// TIA Portal project "SCL EJERCICIO 5" (V11)

(* hardware
DEVICE "S7300/ET200 station_1"  SIMATIC 300-Station
   slot 0: "Perfil soporte_0"  Rail  6ES7 390-1***0-0AA0
   slot 2: "PLC_1"  CPU 313C-2 DP  6ES7 313-6CF03-0AB0  V2.6
      slot 0: "Interfaz MPI_1"  MPI
      slot 1: "Interfaz DP_1"  DP
      slot 2: "DI16/DO16_1"  DI16/DO16
      slot 4: "Contaje_1"  Counter
*)

// ===== PLC "PLC_1"  CPU 313C-2 DP =====

VAR_GLOBAL   // PLC tag table "Tabla de variables estándar"
   "Tag_1" AT %E0.0 : Bool;
   "Tag_2" AT %E0.1 : Bool;
   "Tag_3" AT %E0.2 : Bool;
   "Tag_4" AT %E0.3 : Bool;
   "Tag_5" AT %E0.4 : Bool;
   "Tag_6" AT %E0.5 : Bool;
   "Tag_7" AT %E0.6 : Bool;
   "Tag_8" AT %E0.7 : Bool;
   "Tag_9" AT %E1.0 : Bool;
   "Tag_10" AT %E1.1 : Bool;
   "Tag_11" AT %A0.0 : Bool;
   "Tag_12" AT %A0.1 : Bool;
   "Tag_13" AT %A0.2 : Bool;
   "Tag_14" AT %A0.3 : Bool;
   "Tag_15" AT %A0.4 : Bool;
   "Tag_16" AT %A0.5 : Bool;
   "Tag_17" AT %A0.6 : Bool;
   "Tag_18" AT %A0.7 : Bool;
   "Tag_19" AT %A1.0 : Bool;
   "Tag_20" AT %A1.1 : Bool;
   "Tag_21" AT %M0.0 : Bool;
   "Tag_22" AT %MW10 : Int;
   "Tag_23" AT %A1.2 : Bool;
   "Tag_24" AT %A1.3 : Bool;
   "Tag_25" AT %A2.0 : Bool;
   "Tag_26" AT %T0 : Timer;
   "Tag_27" AT %A2.1 : Bool;
   "Tag_28" AT %A2.2 : Bool;
   "Tag_29" AT %A2.3 : Bool;
   "Tag_30" AT %M0.1 : Bool;
END_VAR

DATA_BLOCK "MEZCLADOR_DB"   // DB2
{ S7_Optimized_Access := 'FALSE' }
VERSION : 0.1
// stored: InstanceOfName MEZCLADOR
"MEZCLADOR"
BEGIN
END_DATA_BLOCK

FUNCTION_BLOCK "MEZCLADOR"   // FB1, SCL
{ S7_Optimized_Access := 'FALSE' }
VERSION : 0.1
   VAR_INPUT
      PRESELECCION : Bool;
      EJECUCION : Bool;
      "SETA EMERGENCIA" : Bool;
      S0 : Bool;
      S1 : Bool;
      S2 : Bool;
      S3 : Bool;
      S4 : Bool;
      S5 : Bool;
      CONTADOR : Int;
   END_VAR
   VAR_OUTPUT
      "MEZCLA 1" : Bool;
      "MEZCLA 2" : Bool;
      "MEZCLA 3" : Bool;
      "MEZCLA 4" : Bool;
      "MEZCLA 5" : Bool;
      "MEZCLA 6" : Bool;
      "VALVULA A" : Bool;
      "VALVULA B" : Bool;
      HOMOGENIZADOR : Bool;
      "VALVULA C" : Bool;
      ENCLAVAMIENTO : Bool;
      REINICIO : Bool;
      contaje : Bool;
      "CONTACTO SETA" : Bool;
   END_VAR
   VAR
      T0 : Bool;
      VISUALIZAR : Time;
      m0 : Bool;
      m1 : Bool;
      t1 : Bool;
      "VISUALIZAR 1" : Time;
   END_VAR
BEGIN
END_FUNCTION_BLOCK

ORGANIZATION_BLOCK "Main"   // OB1, LAD
TITLE = "Main Program Sweep (Cycle)"
{ S7_Optimized_Access := 'FALSE' }
VERSION : 0.1
   VAR_TEMP
      OB1_EV_CLASS : Byte;   // Bits 0-3 = 1 (Coming event), Bits 4-7 = 1 (Event class 1)
      OB1_SCAN_1 : Byte;   // 1 (Cold restart scan 1 of OB 1), 3 (Scan 2-n of OB 1)
      OB1_PRIORITY : Byte;   // Priority of OB Execution
      OB1_OB_NUMBR : Byte;   // 1 (Organization block 1, OB1)
      OB1_RESERVED_1 : Byte;   // Reserved for system
      OB1_RESERVED_2 : Byte;   // Reserved for system
      OB1_PREV_CYCLE : Int;   // Cycle time of previous OB1 scan (milliseconds)
      OB1_MIN_CYCLE : Int;   // Minimum cycle time of OB1 (milliseconds)
      OB1_MAX_CYCLE : Int;   // Maximum cycle time of OB1 (milliseconds)
      OB1_DATE_TIME : Date_And_Time;   // Date and time OB1 started
   END_VAR
   VAR_TEMP   // added for the SCL form of the ladder/FBD networks
      _w1 : Bool;
      _w2 : Bool;
   END_VAR
BEGIN

REGION Network 1
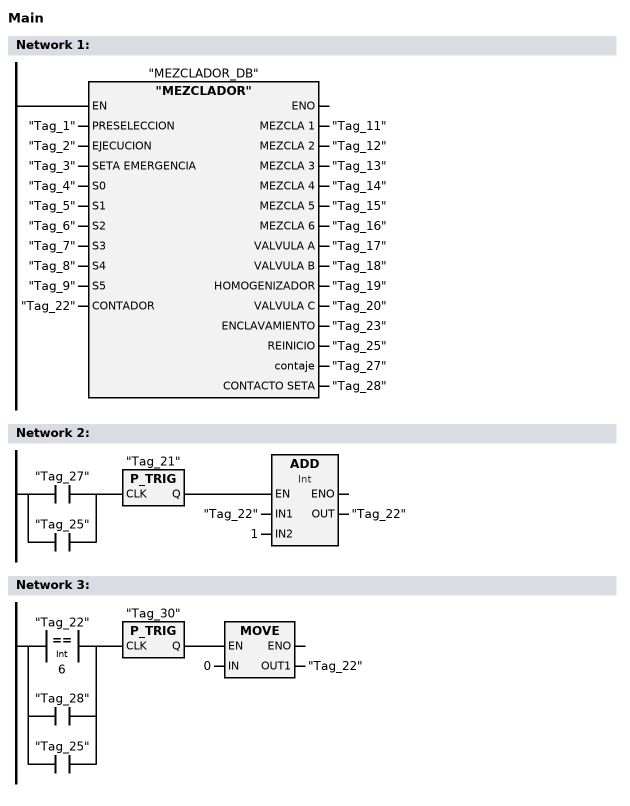
   RUNG wire#powerrail
      "MEZCLADOR_DB"(PRESELECCION := "Tag_1", EJECUCION := "Tag_2", "SETA EMERGENCIA" := "Tag_3", S0 := "Tag_4", S1 := "Tag_5", S2 := "Tag_6", S3 := "Tag_7", S4 := "Tag_8", S5 := "Tag_9", CONTADOR := "Tag_22", "MEZCLA 1" => "Tag_11", "MEZCLA 2" => "Tag_12", "MEZCLA 3" => "Tag_13", "MEZCLA 4" => "Tag_14", "MEZCLA 5" => "Tag_15", "MEZCLA 6" => "Tag_16", "VALVULA A" => "Tag_17", "VALVULA B" => "Tag_18", HOMOGENIZADOR => "Tag_19", "VALVULA C" => "Tag_20", ENCLAVAMIENTO => "Tag_23", REINICIO => "Tag_25", contaje => "Tag_27", "CONTACTO SETA" => "Tag_28")
   END_RUNG
   // the same network as SCL:
   "MEZCLADOR_DB"(PRESELECCION := "Tag_1",   // "MEZCLADOR"
                  EJECUCION := "Tag_2",
                  "SETA EMERGENCIA" := "Tag_3",
                  S0 := "Tag_4",
                  S1 := "Tag_5",
                  S2 := "Tag_6",
                  S3 := "Tag_7",
                  S4 := "Tag_8",
                  S5 := "Tag_9",
                  CONTADOR := "Tag_22",
                  "MEZCLA 1" => "Tag_11",
                  "MEZCLA 2" => "Tag_12",
                  "MEZCLA 3" => "Tag_13",
                  "MEZCLA 4" => "Tag_14",
                  "MEZCLA 5" => "Tag_15",
                  "MEZCLA 6" => "Tag_16",
                  "VALVULA A" => "Tag_17",
                  "VALVULA B" => "Tag_18",
                  HOMOGENIZADOR => "Tag_19",
                  "VALVULA C" => "Tag_20",
                  ENCLAVAMIENTO => "Tag_23",
                  REINICIO => "Tag_25",
                  contaje => "Tag_27",
                  "CONTACTO SETA" => "Tag_28");
END_REGION

REGION Network 2
   RUNG wire#powerrail
      Contact( "Tag_27" )
      wire#w1
      P_Trig( "Tag_21" )
      { S7_Templates := "SrcType := Int"; S7_GenerateENO := "TRUE" } Add(in1 := "Tag_22", in2 := 1, out => "Tag_22")
   END_RUNG
   RUNG wire#powerrail
      Contact( "Tag_25" )
   END_RUNG wire#w1
   // the same network as SCL:
   #_w1 := "Tag_27" OR "Tag_25";
   #_w2 := #_w1 AND NOT "Tag_21";   // rising edge
   "Tag_21" := #_w1;
   IF #_w2 THEN "Tag_22" := "Tag_22" + 1; END_IF;
END_REGION

REGION Network 3
   RUNG wire#powerrail
      { S7_Templates := "SrcType := Int" } EQ_Contact(in1 := "Tag_22", in2 := 6)
      wire#w1
      P_Trig( "Tag_30" )
      { S7_GenerateENO := "TRUE" } Move(in := 0, out1 => "Tag_22")
   END_RUNG
   RUNG wire#powerrail
      Contact( "Tag_28" )
   END_RUNG wire#w1
   RUNG wire#powerrail
      Contact( "Tag_25" )
   END_RUNG wire#w1
   // the same network as SCL:
   #_w1 := ("Tag_22" = 6) OR "Tag_28" OR "Tag_25";
   #_w2 := #_w1 AND NOT "Tag_30";   // rising edge
   "Tag_30" := #_w1;
   IF #_w2 THEN "Tag_22" := 0; END_IF;
END_REGION
END_ORGANIZATION_BLOCK